// TIA Portal V20 export
DATA_BLOCK "DB_Found_Water_Fountain_Functional_Test"   // DB11
{ S7_Optimized_Access := 'TRUE' }
// stored: MemoryReserve 100
   VAR
      Found_Functional_Test : Bool;
      Water_Foutain_Fail_Functional_Test : Bool;
      i : SInt;
      Water_Foutain_Functional_Test : "Functional_Test";
   END_VAR
BEGIN
END_DATA_BLOCK
